SUBAPPLICATION Uebung_004b4d (* Drei gegenseitig verriegelte Toggle-Flip-Flops in einer Kette via AE2-Adapter mit ILOCK_T_FF *)
  (* Standard: 61499-2; Description: Copyright (c) 2023 Meisterschulen am Ostbahnhof This program and the accompanying materials are made available under the terms of the Eclipse Public License 2.0 which is available at https://www.eclipse.org/legal/epl-2.0/ SPDX-License-Identifier: EPL-2.0 *)
  (* Version 1.0, 2023-10-23, Franz Höpfinger, Meisterschulen am Ostbahnhof, initial API and implementation and/or initial documentation *)
  PACKAGE Uebungen;
  IMPORT logiBUS::io::DI::logiBUS_DI::Input_I1;
  IMPORT logiBUS::io::DI::logiBUS_DI::Input_I2;
  IMPORT logiBUS::io::DI::logiBUS_DI::Input_I3;
  IMPORT logiBUS::io::DI::logiBUS_DI_Events::BUTTON_SINGLE_CLICK;
  IMPORT logiBUS::io::DQ::logiBUS_DO::Output_Q1;
  IMPORT logiBUS::io::DQ::logiBUS_DO::Output_Q2;
  IMPORT logiBUS::io::DQ::logiBUS_DO::Output_Q3;
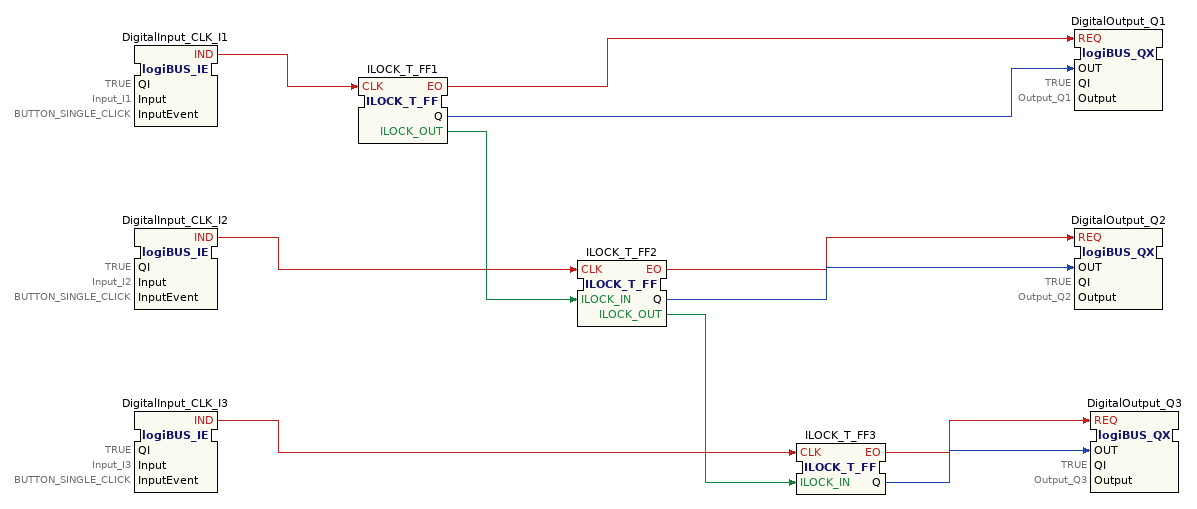
  (* durch den Einsatz eines Bidirektionalen Adapters: 1 Verbindung REICHT ! *)
  FBS
    DigitalOutput_Q1 : logiBUS::io::DQ::logiBUS_QX(QI := TRUE, Output := Output_Q1);
    DigitalInput_CLK_I1 : logiBUS::io::DI::logiBUS_IE(QI := TRUE, Input := Input_I1, InputEvent := BUTTON_SINGLE_CLICK);
    DigitalOutput_Q2 : logiBUS::io::DQ::logiBUS_QX(QI := TRUE, Output := Output_Q2);
    DigitalInput_CLK_I2 : logiBUS::io::DI::logiBUS_IE(QI := TRUE, Input := Input_I2, InputEvent := BUTTON_SINGLE_CLICK);
    ILOCK_T_FF1 : logiBUS::signalprocessing::interlock::ILOCK_T_FF;
    ILOCK_T_FF2 : logiBUS::signalprocessing::interlock::ILOCK_T_FF;
    ILOCK_T_FF3 : logiBUS::signalprocessing::interlock::ILOCK_T_FF;
    DigitalOutput_Q3 : logiBUS::io::DQ::logiBUS_QX(QI := TRUE, Output := Output_Q3);
    DigitalInput_CLK_I3 : logiBUS::io::DI::logiBUS_IE(QI := TRUE, Input := Input_I3, InputEvent := BUTTON_SINGLE_CLICK);
  END_FBS
  EVENT_CONNECTIONS
    DigitalInput_CLK_I1.IND TO ILOCK_T_FF1.CLK;
    DigitalInput_CLK_I2.IND TO ILOCK_T_FF2.CLK;
    DigitalInput_CLK_I3.IND TO ILOCK_T_FF3.CLK;
    ILOCK_T_FF1.EO TO DigitalOutput_Q1.REQ;
    ILOCK_T_FF2.EO TO DigitalOutput_Q2.REQ;
    ILOCK_T_FF3.EO TO DigitalOutput_Q3.REQ;
  END_CONNECTIONS
  DATA_CONNECTIONS
    ILOCK_T_FF1.Q TO DigitalOutput_Q1.OUT;
    ILOCK_T_FF2.Q TO DigitalOutput_Q2.OUT;
    ILOCK_T_FF3.Q TO DigitalOutput_Q3.OUT;
  END_CONNECTIONS
  ADAPTER_CONNECTIONS
    ILOCK_T_FF1.ILOCK_OUT TO ILOCK_T_FF2.ILOCK_IN;
    ILOCK_T_FF2.ILOCK_OUT TO ILOCK_T_FF3.ILOCK_IN;
  END_CONNECTIONS
END_SUBAPPLICATION
